{attribute 'qualified_only'}
VAR_GLOBAL
	ActuatorPivot : ST_Coordinates := (Height:=2610.7, Distance:=-1036.01); //Zero angle coordinates
	BenchPivot : ST_Coordinates := (Height:=1386.7, Distance:=-837); //Zero angle coordinates
	FloatPivot : ST_Coordinates := (Height:=2936.7, Distance:=-691.5); //Zero angle coordinates
	SamplePivot : ST_Coordinates := (Height:=0, Distance:=0);
	
	SampleToBench_Lever : LREAL; //READ ONLY
	SampleToBench_Angle : LREAL; //READ ONLY
	
	BenchToFloat_Lever : LREAL; //READ ONLY
	BenchToFloat_Angle : LREAL; //READ ONLY
	BenchToActuator_Angle : LREAL; //READ ONLY
	
	BenchPivotTarget : ST_Coordinates;
END_VAR

(* stored: Version 1.1.0.1, ProductVersion 3.1.4026.12
   GVL KinematicConstants: Id {5094f862-43b2-4615-b739-9acf28055e9d} *)
